// TwinCAT 3 PLC project TcoAimTtiPowerSupply
// Title: TcoAimTtiPowerSupply
// Company: Vortex.Library
// Author: TcOpenGroup
// ProjectVersion: 0.6.0.913
// ProgramVersion: 3.1.4026.12
// libraries:
//   Tc2_MC2, * (Beckhoff Automation GmbH)
//   Tc2_MC2_Drive, * (Beckhoff Automation GmbH)
//   Tc2_Standard, * (Beckhoff Automation GmbH)
//   Tc2_System, * (Beckhoff Automation GmbH)
//   Tc3_Module, * (Beckhoff Automation GmbH)
//   TcoAbstractions, 0.6.0.913 (Vortex.Library)
//   TcoCore, 0.6.0.913 (Vortex.Library)
//   TcoIo, 0.6.0.913 (Vortex.Library)
//   TcoUtilities, 0.6.0.913 (Vortex.Library)
// project tree:
//   DUTs/ TcoQlSeriesSupply_Config_v_1_x_x.TcDUT (not stored), TcoQlSeriesSupply_GetControl_v_1_x_x.TcDUT (not stored), TcoQlSeriesSupply_SetControl_v_1_x_x.TcDUT (not stored), TcoQlSeriesSupply_State_v_1_x_x.TcDUT (not stored), TcoQlSeriesSupply_Status_v_1_x_x.TcDUT (not stored)
//   / PlcTask.TcTTO (not stored)
//   POUs/ MAIN.TcPOU (not stored)
//   POUs/Prototypes/Command/ TcoQlGetCommandTask.TcPOU (not stored), TcoQlSetCommandTask.TcPOU (not stored), TcoQlSeriesSupplyTask.TcPOU (not stored)
//   POUs/Prototypes/QLSeries/ TcoQl355P_v_1_x_x.TcPOU (not stored)
//   POUs/Prototypes/Structs/ eTcoQWlSeriesSupplyGetCommands_v_1_x_x.TcDUT, eTcoQWlSeriesSupplySetCommands_v_1_x_x.TcDUT (not stored)
// real-time tasks:
//   TASK PlcTask: cycle T#10ms, priority 20, ADS port 350
//   TASK PlcTask1: cycle T#10ms, priority 1, ADS port 351
//   TASK PN: cycle T#8ms, priority 2, ADS port 301
// motion (NC):
//   TASK NC-Task 1 SAF: cycle T#2ms, priority 4, ADS port 501
//   TASK NC-Task 1 SVB: cycle T#10ms, priority 8, ADS port 511
//   AXIS Axis 1 (id 1)
//     Dynamic: Acceleration=5979.5, Deceleration=5979.5, Jerk=17938.5
//     Velo: RefSearch=39.8633642666667, RefSync=39.8633642666667, SlowManual=199.316821333333, FastManual=1195.900928, Fast=3986.33642666667, Maximum=3986.34
//     OtherSettings: AllowMotionCmdToSlave=true
//     encoder EncType=1
//       EncPara: ScaleFactorNumerator=104.8576, ScaleFactorDenominator=1048576, Offset=-0.001200000000608
//     drive DrvType=5
//       Analog: VeloReferenz=4384.97006933333, TorqueSetpointScale=10, ScaleFactorActTorque=0.1
//       TimeComp: TaskDelayCycles=1
//     controller CtrType=1
//       CtrPara: PriorControlFactor=1
//         Observer: BandWidth=20
//   AXIS Axis 2 (id 2)
//     Dynamic: Acceleration=500, Deceleration=500, Jerk=1000
//     Velo: SlowManual=10, FastManual=50, Maximum=3986.34
//     OtherSettings: AllowMotionCmdToSlave=true
//     encoder EncType=1
//       EncPara: ScaleFactorNumerator=1, ScaleFactorDenominator=1024
//     drive DrvType=5
//       Analog: VeloReferenz=4384.97006933333, TorqueSetpointScale=10, ScaleFactorActTorque=0.1
//       TimeComp: TaskDelayCycles=1
//     controller CtrType=1
//       CtrPara: PriorControlFactor=1
//         PosDiffControl: Enable=false
//         PID: PosKp=0.1
//         Observer: BandWidth=20
//   AXIS Axis 3 (id 3)
//     Dynamic: Acceleration=500, Deceleration=500, Jerk=1000
//     Velo: SlowManual=10, FastManual=50, Maximum=3986.34
//     OtherSettings: AllowMotionCmdToSlave=true
//     encoder EncType=1
//       EncPara: ScaleFactorNumerator=1, ScaleFactorDenominator=1024
//     drive DrvType=5
//       Analog: VeloReferenz=4384.97006933333, TorqueSetpointScale=10, ScaleFactorActTorque=0.1
//       TimeComp: TaskDelayCycles=1
//     controller CtrType=1
//       CtrPara: PriorControlFactor=1
//         PosDiffControl: Enable=false
//         PID: PosKp=0.1
//         Observer: BandWidth=20
//   AXIS Axis 4 (id 4)
//     Dynamic: Acceleration=500, Deceleration=500, Jerk=1000
//     Velo: SlowManual=10, FastManual=50, Maximum=3986.34
//     OtherSettings: AllowMotionCmdToSlave=true
//     encoder EncType=1
//       EncPara: ScaleFactorNumerator=1, ScaleFactorDenominator=1024
//     drive DrvType=5
//       Analog: VeloReferenz=4384.97006933333, TorqueSetpointScale=10, ScaleFactorActTorque=0.1
//       TimeComp: TaskDelayCycles=1
//     controller CtrType=1
//       CtrPara: PriorControlFactor=1
//         PosDiffControl: Enable=false
//         PID: PosKp=0.1
//         Observer: BandWidth=20
// I/O:
//   DEVICE Device 4 (EtherCAT) (disabled), AmsNetId 172.20.10.104.5.1
//     Term 1 (EK1100) [EK1100 EtherCAT Coupler (2A E-Bus)]
//       Term 2 (EL1008) [EL1008 8Ch. Dig. Input 24V, 3ms]
//       Term 3 (EL2008) [EL2008 8Ch. Dig. Output 24V, 0.5A]
//       Term 4 (EL3052) [EL3052 2Ch. Ana. Input 4-20mA]
//       Term 5 (EL9576) [EL9576 Brake chopper terminal]
//       Term 6 (EL7211-0010) [EL7211-0010 1Ch. MDP742 Servo motor output stage with OCT (50V, 4.5A RMS)]
//       Term 14 (EL7047) [EL7047 1Ch. Stepper motor output stage (50V, 5A)]
//       Term 8 (EL9011) [EL9011 End Terminal]
//   DEVICE Device 1 (EtherCAT) (disabled), AmsNetId 192.168.4.1.2.1
//     Drive 7 (IndraDrive MPB20) [IndraDrive MPB20]
//   DEVICE Device 2 (EtherCAT) (disabled), AmsNetId 192.168.4.1.3.1
//     Term 1 (EK1200) [EK1200-5000 EtherCAT Power supply (2A E-Bus)]
//       Term 10 (EK1122) [EK1122 2 port EtherCAT junction]
//       Term 13 (EL6631) [EL6631 PROFINET IO Controller]
//       Term 12 (EL1809) [EL1809 16Ch. Dig. Input 24V, 3ms]
//       Term 13 (EL2809) [EL2809 16Ch. Dig. Output 24V, 0.5A]
//       Term 15 (EL4004) [EL4004 4Ch. Ana. Output 0-10V, 12bit]
//       Term 16 (EL7342) [EL7342 2Ch. DC motor output stage (50V, 3.5A)]
//       Term 17 (EL4004) [EL4004 4Ch. Ana. Output 0-10V, 12bit]
//       Term 18 (EL6001) [EL6001 Interface (RS232)]
//       Term 10 (EL9011) [EL9011 End Terminal]
//   DEVICE Device 3 (EL6631) (disabled), AmsNetId 192.168.4.1.4.1
//     robot1 [ABB Robotics The robot controller's internal PROFINET IO device. 888-3] (disabled)
//       modules: Term 1 (DAP Module), Term 2 (DI 64 bytes), Term 3 (DO 64 bytes)
//     robot2 [ABB Robotics The OmniCore controller's internal PROFINET IO device. 3020-x]
//       modules: Term 7 (DAP Module), Term 8 (DI 64 bytes), Term 9 (DO 64 bytes)

// ---- POUs/Prototypes/Structs/eTcoQWlSeriesSupplyGetCommands_v_1_x_x.TcDUT
{attribute 'qualified_only'}
{attribute 'strict'}
TYPE
    eTcoQWlSeriesSupplyGetCommands_v_1_x_x :
    (
		//Instrument Specific Commands
		V	:=1,
		I	:=2,
		OVP	:=3,
		OCP	:=4,
		VO	:=5,
		IO	:=6,
		RANGE :=7,
		DELTAV:=8,
		DELTAI:=9,
		OP:=10,
        LSR :=11,
		LSE:=12,
		
		//System and Status Commands
		EER:=22,
		QER:=23, 
		ESE:=24, 
		ESR:=25,
		IST:=26,
		OPC:=27,
		PRE:=28,
		SRE:=29, 
		STB:=30, 
		
		//Interface Management Commands
		IFLOCK:=41,
		ADDRESS:=42,
		IPADDR:=43, 
		NETMASK:=44,
		NETCONFIG:=45,
		
		//Miscellaneous Commands
		IDN:=70,
		TST:=71
		

    );
END_TYPE
